{attribute 'qualified_only'}
VAR_GLOBAL
	hwAirDataIN : stAi4CH;
END_VAR

(* stored: Version 1.1.0.1, ProductVersion 3.1.4024.2
   GVL IO: Id {c0227015-dc69-4708-8625-cedcbecd4015} *)
